// TIA Portal project "SistemaSemaforico" (V15.1)

(* hardware
DEVICE "S7-1200 station_1"  S7-1200 Station
   slot 0: "Telaio di montaggio_0"  S7-1200 Rack  Rack  V1.0
   slot 1: "PLC_1"  CPU 1214C DC/DC/DC  6ES7 214-1AG40-0XB0  V4.2
*)

// ===== PLC "PLC_1"  CPU 1214C DC/DC/DC =====

VAR_GLOBAL   // PLC tag table "Tabella delle variabili standard"
   "Abilita" AT %I0.0 : Bool;
   "V1" AT %Q0.0 : Bool;
   "V2" AT %Q0.1 : Bool;
   "G1" AT %Q0.2 : Bool;
   "G2" AT %Q0.3 : Bool;
   "R1" AT %Q0.4 : Bool;
   "R2" AT %Q0.5 : Bool;
   "Pedone" AT %M0.0 : Bool;
   "Mutex" AT %M0.1 : Bool;
   "P" AT %I0.1 : Bool;
END_VAR

VAR_GLOBAL CONSTANT   // PLC tag table "Tabella delle variabili standard"
   "DurataVerde" : Time := T#55s;
   "DurataGiallo" : Time := T#5s;
   "DurataRosso" : Time := T#60s;
END_VAR

TYPE "StatoSemaforo"
   STRUCT
      Home : Bool := true;
      Rosso : Bool;
      Verde : Bool;
      Giallo : Bool;
   END_STRUCT;
END_TYPE

DATA_BLOCK "Semaforo_DB"   // DB1
{ S7_Optimized_Access := 'TRUE' }
VERSION : 0.1
// stored: InstanceOfName Semaforo
"Semaforo"
BEGIN
END_DATA_BLOCK

DATA_BLOCK "Semaforo_DB_1"   // DB2
{ S7_Optimized_Access := 'TRUE' }
VERSION : 0.1
// stored: InstanceOfName Semaforo
"Semaforo"
BEGIN
END_DATA_BLOCK

FUNCTION_BLOCK "Semaforo"   // FB1, LAD
{ S7_Optimized_Access := 'TRUE' }
VERSION : 0.1
   VAR_INPUT
      Abilita : Bool;
      DurataVerde : Time;
      DurataGiallo : Time;
      DurataRosso : Time;
   END_VAR
   VAR_OUTPUT
      Verde : Bool;
      Giallo : Bool;
      Rosso : Bool;
   END_VAR
   VAR_IN_OUT
      Mutex : Bool;
   END_VAR
   VAR RETAIN
      Stato : "StatoSemaforo";
      IEC_Timer_0_Instance : TON_TIME;
      IEC_Timer_0_Instance_1 : TON_TIME;
      IEC_Timer_0_Instance_2 : TON_TIME;
      PadroneMutex : Bool;
   END_VAR
   VAR_TEMP   // added for the SCL form of the ladder/FBD networks
      _w1 : Bool;
   END_VAR
BEGIN

REGION Network 1
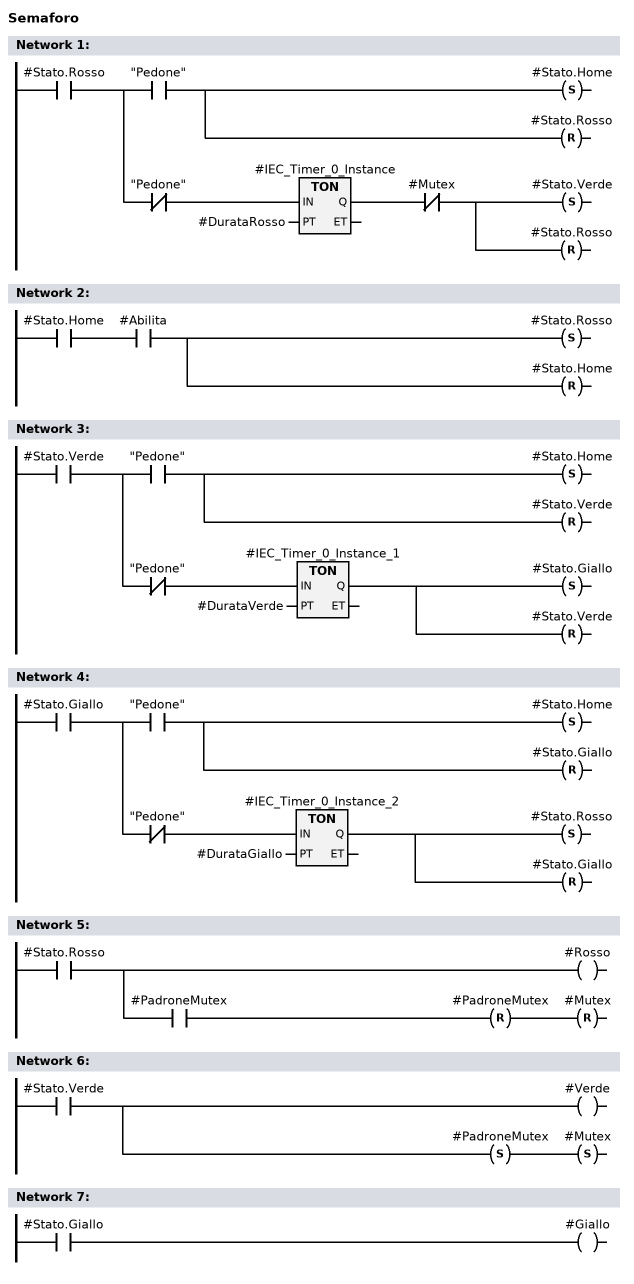
   IF #Stato.Rosso AND "Pedone" THEN #Stato.Home := TRUE; END_IF;
   #_w1 := #Stato.Rosso;
   IF #Stato.Rosso AND "Pedone" THEN #Stato.Rosso := FALSE; END_IF;
   #IEC_Timer_0_Instance(IN := #_w1 AND NOT "Pedone", PT := #DurataRosso);   // TON
   IF #IEC_Timer_0_Instance.Q AND NOT #Mutex THEN
       #Stato.Verde := TRUE;
       #Stato.Rosso := FALSE;
   END_IF;
END_REGION

REGION Network 2
   RUNG wire#powerrail
      Contact( #Stato.Home )
      Contact( #Abilita )
      wire#w1
      S_Coil( #Stato.Rosso )
   END_RUNG
   RUNG wire#w1
      R_Coil( #Stato.Home )
   END_RUNG
   // the same network as SCL:
   IF #Stato.Home AND #Abilita THEN
       #Stato.Rosso := TRUE;
       #Stato.Home := FALSE;
   END_IF;
END_REGION

REGION Network 3
   IF #Stato.Verde AND "Pedone" THEN #Stato.Home := TRUE; END_IF;
   #_w1 := #Stato.Verde;
   IF #Stato.Verde AND "Pedone" THEN #Stato.Verde := FALSE; END_IF;
   #IEC_Timer_0_Instance_1(IN := #_w1 AND NOT "Pedone", PT := #DurataVerde);   // TON
   IF #IEC_Timer_0_Instance_1.Q THEN
       #Stato.Giallo := TRUE;
       #Stato.Verde := FALSE;
   END_IF;
END_REGION

REGION Network 4
   IF #Stato.Giallo AND "Pedone" THEN #Stato.Home := TRUE; END_IF;
   #_w1 := #Stato.Giallo;
   IF #Stato.Giallo AND "Pedone" THEN #Stato.Giallo := FALSE; END_IF;
   #IEC_Timer_0_Instance_2(IN := #_w1 AND NOT "Pedone", PT := #DurataGiallo);   // TON
   IF #IEC_Timer_0_Instance_2.Q THEN
       #Stato.Rosso := TRUE;
       #Stato.Giallo := FALSE;
   END_IF;
END_REGION

REGION Network 5
   RUNG wire#powerrail
      Contact( #Stato.Rosso )
      wire#w1
      Coil( #Rosso )
   END_RUNG
   RUNG wire#w1
      Contact( #PadroneMutex )
      R_Coil( #PadroneMutex )
      R_Coil( #Mutex )
   END_RUNG
   // the same network as SCL:
   #Rosso := #Stato.Rosso;
   #_w1 := #Stato.Rosso AND #PadroneMutex;
   IF #_w1 THEN
       #PadroneMutex := FALSE;
       #Mutex := FALSE;
   END_IF;
END_REGION

REGION Network 6
   RUNG wire#powerrail
      Contact( #Stato.Verde )
      wire#w1
      Coil( #Verde )
   END_RUNG
   RUNG wire#w1
      S_Coil( #PadroneMutex )
      S_Coil( #Mutex )
   END_RUNG
   // the same network as SCL:
   #Verde := #Stato.Verde;
   IF #Stato.Verde THEN
       #PadroneMutex := TRUE;
       #Mutex := TRUE;
   END_IF;
END_REGION

REGION Network 7
   RUNG wire#powerrail
      Contact( #Stato.Giallo )
      Coil( #Giallo )
   END_RUNG
   // the same network as SCL:
   #Giallo := #Stato.Giallo;
END_REGION
END_FUNCTION_BLOCK

ORGANIZATION_BLOCK "Main"   // OB1, LAD, ProgramCycle
TITLE = "Main Program Sweep (Cycle)"
{ S7_Optimized_Access := 'TRUE' }
VERSION : 0.1
   VAR_INPUT
      Initial_Call : Bool;   // Initial call of this OB
      Remanence : Bool;   // =True, if remanent data are available
   END_VAR
BEGIN

REGION Network 1
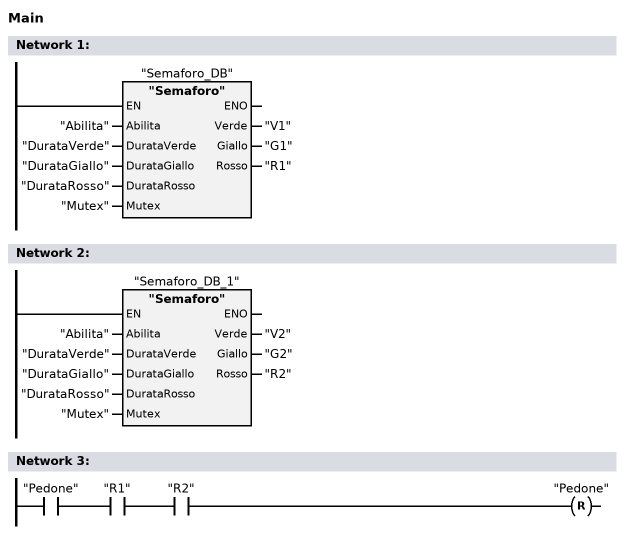
   RUNG wire#powerrail
      "Semaforo_DB"(Abilita := "Abilita", DurataVerde := "DurataVerde", DurataGiallo := "DurataGiallo", DurataRosso := "DurataRosso", Mutex := "Mutex", Verde => "V1", Giallo => "G1", Rosso => "R1")
   END_RUNG
   // the same network as SCL:
   "Semaforo_DB"(Abilita := "Abilita",   // "Semaforo"
                 DurataVerde := "DurataVerde",
                 DurataGiallo := "DurataGiallo",
                 DurataRosso := "DurataRosso",
                 Mutex := "Mutex",
                 Verde => "V1",
                 Giallo => "G1",
                 Rosso => "R1");
END_REGION

REGION Network 2
   RUNG wire#powerrail
      "Semaforo_DB_1"(Abilita := "Abilita", DurataVerde := "DurataVerde", DurataGiallo := "DurataGiallo", DurataRosso := "DurataRosso", Mutex := "Mutex", Verde => "V2", Giallo => "G2", Rosso => "R2")
   END_RUNG
   // the same network as SCL:
   "Semaforo_DB_1"(Abilita := "Abilita",   // "Semaforo"
                   DurataVerde := "DurataVerde",
                   DurataGiallo := "DurataGiallo",
                   DurataRosso := "DurataRosso",
                   Mutex := "Mutex",
                   Verde => "V2",
                   Giallo => "G2",
                   Rosso => "R2");
END_REGION

REGION Network 3
   RUNG wire#powerrail
      Contact( "Pedone" )
      Contact( "R1" )
      Contact( "R2" )
      R_Coil( "Pedone" )
   END_RUNG
   // the same network as SCL:
   IF "Pedone" AND "R1" AND "R2" THEN "Pedone" := FALSE; END_IF;
END_REGION
END_ORGANIZATION_BLOCK

ORGANIZATION_BLOCK "SettaPedone"   // OB40, LAD, HWProcessInterrupt
{ S7_Optimized_Access := 'TRUE' }
VERSION : 0.1
   VAR_INPUT
      LADDR : Hw_Io;   // Hardware identifier
      USI : Word;   // User structure identifier
      IChannel : USInt;   // Interrupt channel number
      EventType : Byte;   // EventType
   END_VAR
BEGIN

REGION Network 1
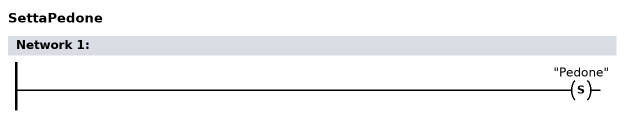
   RUNG wire#powerrail
      S_Coil( "Pedone" )
   END_RUNG
   // the same network as SCL:
   "Pedone" := TRUE;
END_REGION
END_ORGANIZATION_BLOCK